PROGRAM MAIN
VAR
	i: INT;
END_VAR

 PLC_PRG();

END_PROGRAM

(* stored: Version 1.1.0.1, ProductVersion 3.1.4022.12
   POU MAIN: Id {720f5241-2610-4e42-b247-84b15ca27248}, SpecialFunc None *)
